// Mitsubishi GX Works2 project: stepper_jog_speed_pos   PLC: FX1S

PROGRAM MAIN
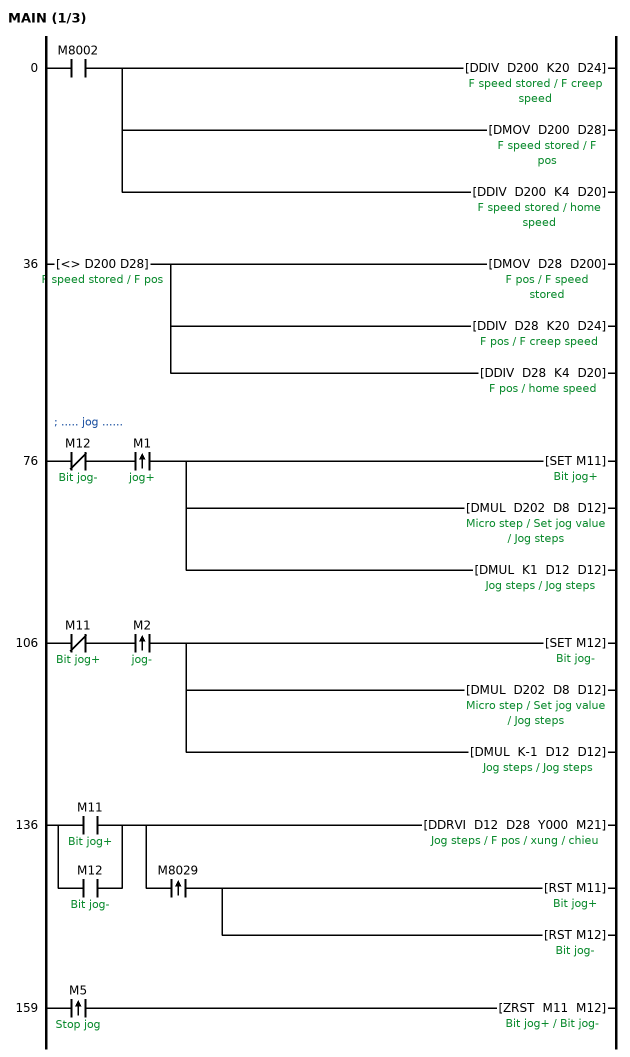
0     LD      M8002
      DDIV    D200 K20 D24  ; F speed stored / F creep speed
      DMOV    D200 D28  ; F pos
      DDIV    D200 K4 D20  ; home speed
36    LD<>    D200 D28  ; F speed stored / F pos
      DMOV    D28 D200
      DDIV    D28 K20 D24
      DDIV    D28 K4 D20
; ..... jog ......
76    LDI     M12  ; Bit jog-
      ANDP    M1  ; jog+
      SET     M11  ; Bit jog+
      DMUL    D202 D8 D12  ; Micro step / Set jog value / Jog steps
      DMUL    K1 D12 D12
106   LDI     M11  ; Bit jog+
      ANDP    M2  ; jog-
      SET     M12  ; Bit jog-
      DMUL    D202 D8 D12
      DMUL    K-1 D12 D12
136   LD      M11  ; Bit jog+
      OR      M12  ; Bit jog-
      DDRVI   D12 D28 Y000 M21  ; xung / chieu
      ANDP    M8029
      RST     M11  ; Bit jog+
      RST     M12  ; Bit jog-
159   LDP     M5  ; Stop jog
      ZRST    M11 M12
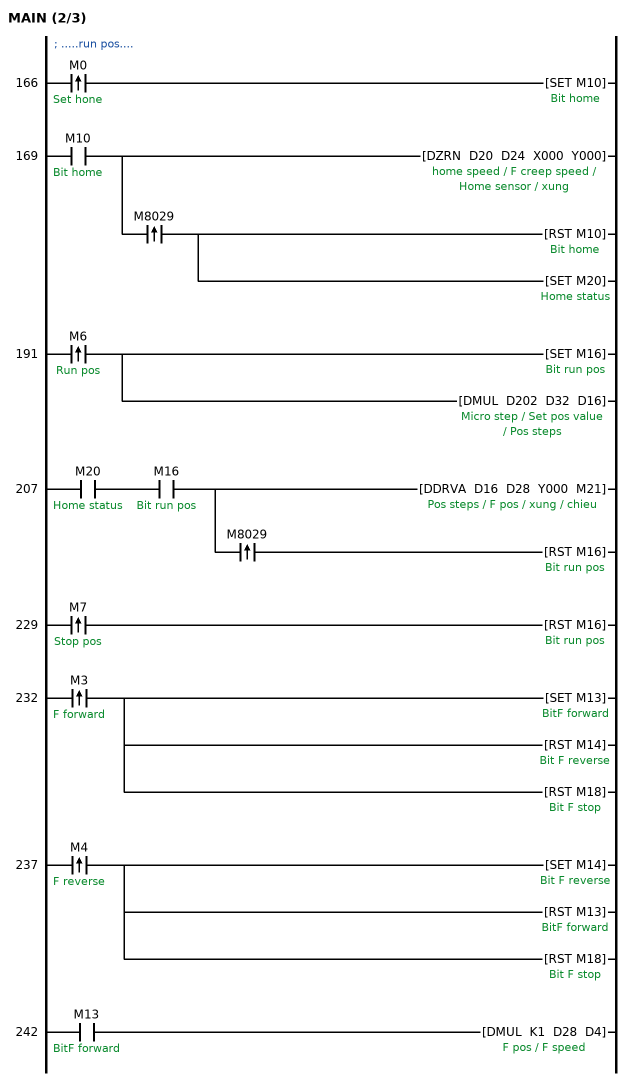
; .....run pos....
166   LDP     M0  ; Set hone
      SET     M10  ; Bit home
169   LD      M10  ; Bit home
      DZRN    D20 D24 X000 Y000  ; Home sensor
      ANDP    M8029
      RST     M10  ; Bit home
      SET     M20  ; Home status
; 
191   LDP     M6  ; Run pos
      SET     M16  ; Bit run pos
      DMUL    D202 D32 D16  ; Set pos value / Pos steps
207   LD      M20  ; Home status
      AND     M16  ; Bit run pos
      DDRVA   D16 D28 Y000 M21
      ANDP    M8029
      RST     M16  ; Bit run pos
229   LDP     M7  ; Stop pos
      RST     M16  ; Bit run pos
232   LDP     M3  ; F forward
      SET     M13  ; BitF forward
      RST     M14  ; Bit F reverse
      RST     M18  ; Bit F stop
237   LDP     M4  ; F reverse
      SET     M14  ; Bit F reverse
      RST     M13  ; BitF forward
      RST     M18  ; Bit F stop
242   LD      M13  ; BitF forward
      DMUL    K1 D28 D4  ; F speed
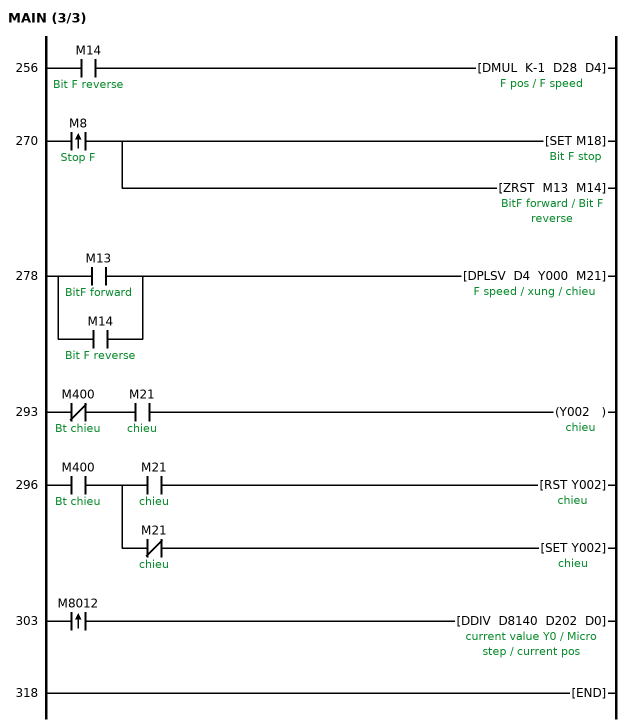
256   LD      M14  ; Bit F reverse
      DMUL    K-1 D28 D4
270   LDP     M8  ; Stop F
      SET     M18  ; Bit F stop
      ZRST    M13 M14
278   LD      M13  ; BitF forward
      OR      M14  ; Bit F reverse
      DPLSV   D4 Y000 M21
293   LDI     M400  ; Bt chieu
      AND     M21  ; chieu
      OUT     Y002  ; chieu
296   LD      M400  ; Bt chieu
      MPS
      AND     M21  ; chieu
      RST     Y002  ; chieu
      MPP
      ANI     M21  ; chieu
      SET     Y002  ; chieu
303   LDP     M8012
      DDIV    D8140 D202 D0  ; current value Y0 / current pos
318   END
END_PROGRAM

// device comments not shown above
Y003  ; enable
M17  ; Bit stop pos
